SYSTEM CNV_LOOP_2_mess (* System Configuration *)
  (* Standard: 61499-1 *)
  (* Version 0.4, 2009-03-05, JHC, Holobloc Inc., Deleted Application. *)
  (* Version 0.3, 2003-12-05, JHC, Rockwell Automation, Renamed from NEWSYSTEM. *)
  (* Version 0.2, 2002-11-05, JHC, Rockwell Automation, Fixed missing (empty) FBD in Application. *)
  (* Version 0.1, 2002-01-17, JHC, Rockwell Automation, Minor cleanup *)
  (* Version 0.0, 2000-05-27, JHC, Rockwell Automation *)
  DEVICE HMI : FRAME_DEVICE(BOUNDS := [0,0,200,300], GRID := [10,10])
    RESOURCE CNV1_HMI : PANEL_RESOURCE
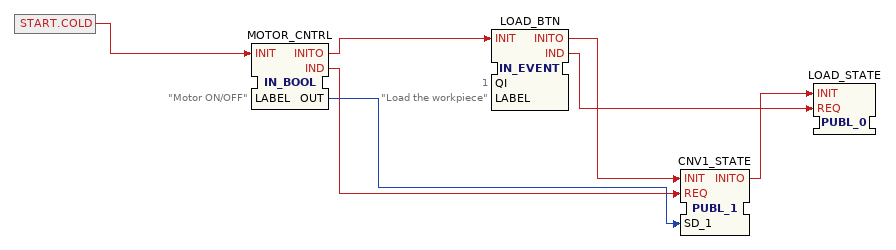
      FBS
        MOTOR_CNTRL : IN_BOOL(LABEL := "Motor ON/OFF");
        LOAD_BTN : IN_EVENT(QI := 1, LABEL := "Load the workpiece");
        LOAD_STATE : PUBL_0;
        CNV1_STATE : PUBL_1;
      END_FBS
      EVENT_CONNECTIONS
        START.COLD TO MOTOR_CNTRL.INIT;
        MOTOR_CNTRL.INITO TO LOAD_BTN.INIT;
        LOAD_BTN.INITO TO CNV1_STATE.INIT;
        CNV1_STATE.INITO TO LOAD_STATE.INIT;
        LOAD_BTN.IND TO LOAD_STATE.REQ;
        MOTOR_CNTRL.IND TO CNV1_STATE.REQ;
      END_CONNECTIONS
      DATA_CONNECTIONS
        MOTOR_CNTRL.OUT TO CNV1_STATE.SD_1;
      END_CONNECTIONS
    END_RESOURCE
  END_DEVICE
  DEVICE MODEL : FRAME_DEVICE(BOUNDS := [0,0,200,300])
    RESOURCE CNV1_MODEL : PANEL_RESOURCE
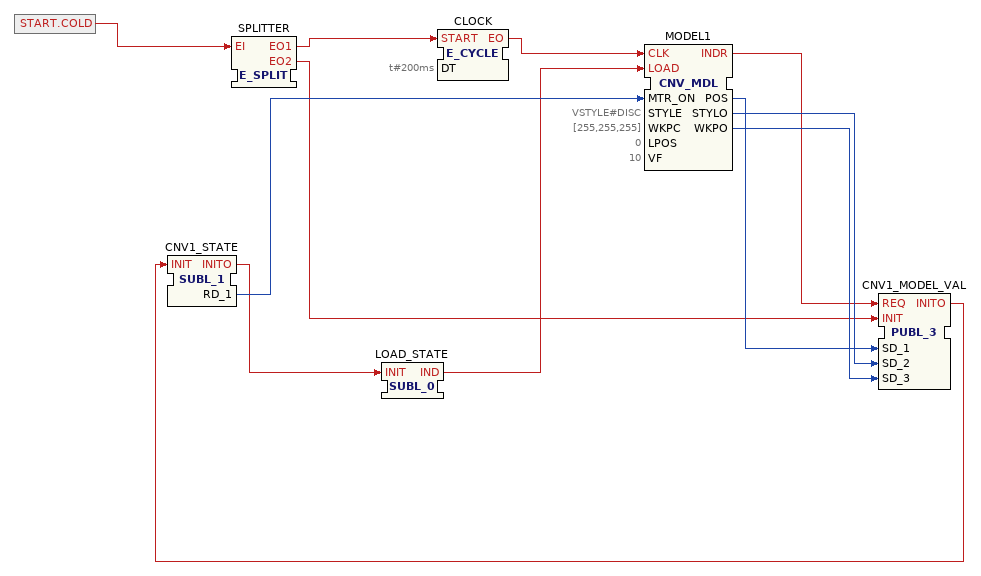
      FBS
        CLOCK : E_CYCLE(DT := t#200ms);
        MODEL1 : CNV_MDL(STYLE := VSTYLE#DISC, WKPC := [255,255,255], LPOS := 0, VF := 10);
        SPLITTER : E_SPLIT;
        CNV1_MODEL_VAL : PUBL_3;
        LOAD_STATE : SUBL_0;
        CNV1_STATE : SUBL_1;
      END_FBS
      EVENT_CONNECTIONS
        CLOCK.EO TO MODEL1.CLK;
        START.COLD TO SPLITTER.EI;
        SPLITTER.EO1 TO CLOCK.START;
        MODEL1.INDR TO CNV1_MODEL_VAL.REQ;
        SPLITTER.EO2 TO CNV1_MODEL_VAL.INIT;
        CNV1_MODEL_VAL.INITO TO CNV1_STATE.INIT;
        CNV1_STATE.INITO TO LOAD_STATE.INIT;
        LOAD_STATE.IND TO MODEL1.LOAD;
      END_CONNECTIONS
      DATA_CONNECTIONS
        MODEL1.POS TO CNV1_MODEL_VAL.SD_1;
        MODEL1.STYLO TO CNV1_MODEL_VAL.SD_2;
        MODEL1.WKPO TO CNV1_MODEL_VAL.SD_3;
        CNV1_STATE.RD_1 TO MODEL1.MTR_ON;
      END_CONNECTIONS
    END_RESOURCE
    RESOURCE CLK_MODEL : PANEL_RESOURCE
    END_RESOURCE
  END_DEVICE
  DEVICE VIEW : FRAME_DEVICE(BOUNDS := [200,0,300,300])
    RESOURCE VIEW_Resource : VIEW_PANEL(DIA := 20, SIZE := [15,15])
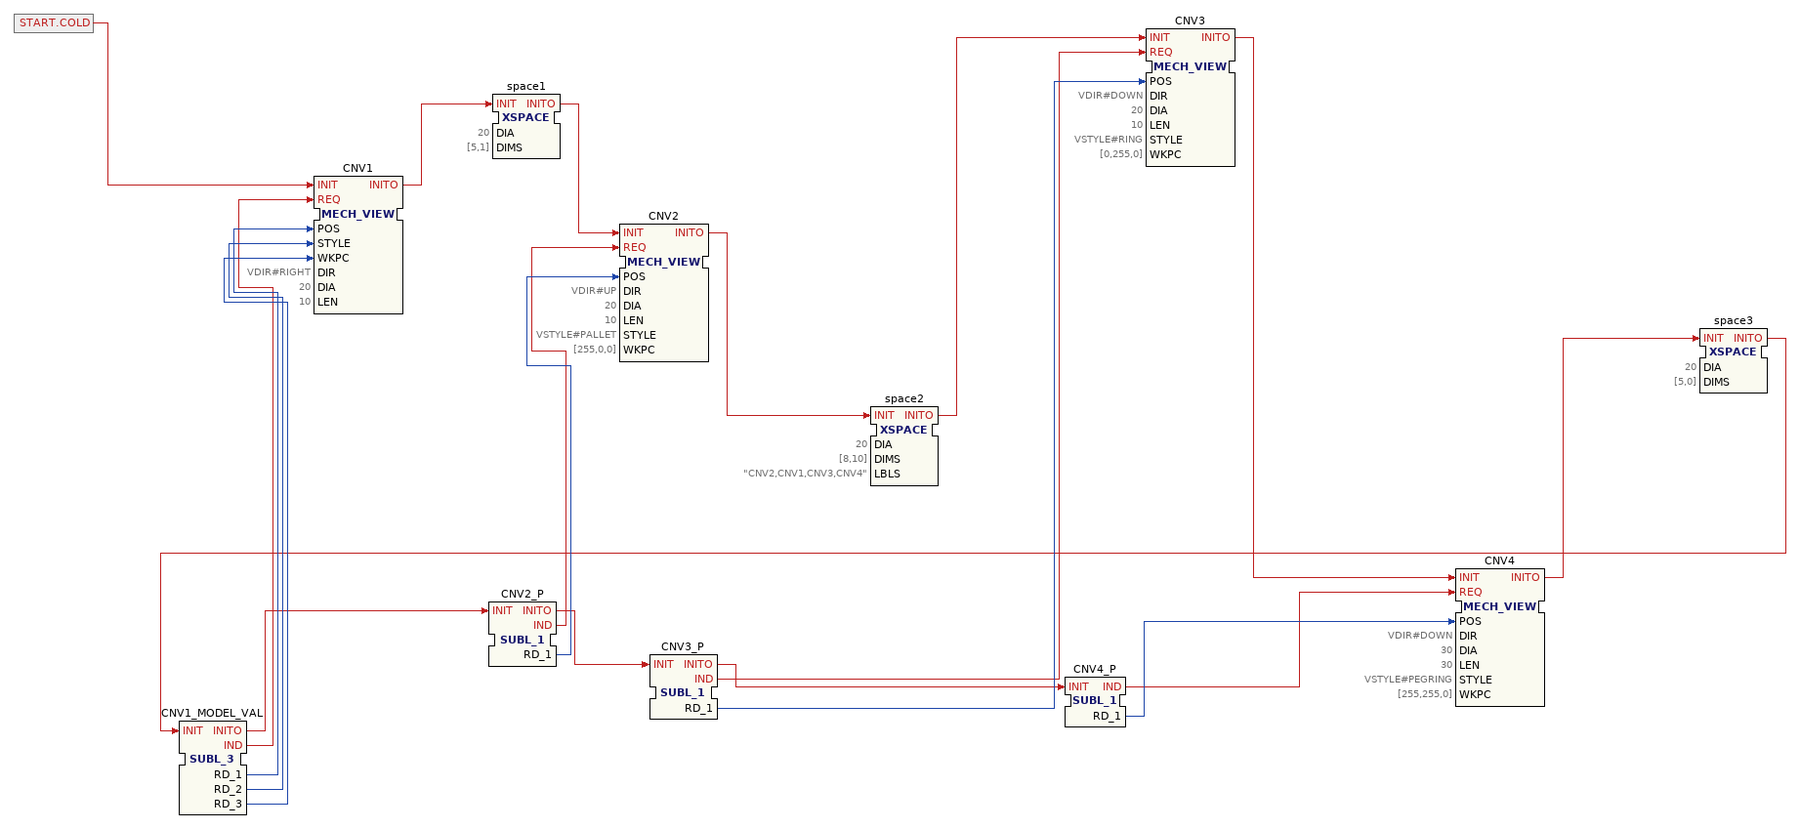
      FBS
        CNV1 : MECH_VIEW(DIR := VDIR#RIGHT, DIA := 20, LEN := 10);
        CNV2 : MECH_VIEW(DIR := VDIR#UP, DIA := 20, LEN := 10, STYLE := VSTYLE#PALLET, WKPC := [255,0,0]);
        CNV3 : MECH_VIEW(DIR := VDIR#DOWN, DIA := 20, LEN := 10, STYLE := VSTYLE#RING, WKPC := [0,255,0]);
        CNV4 : MECH_VIEW(DIR := VDIR#DOWN, DIA := 30, LEN := 30, STYLE := VSTYLE#PEGRING, WKPC := [255,255,0]);
        space1 : XSPACE(DIA := 20, DIMS := [5,1]);
        space2 : XSPACE(DIA := 20, DIMS := [8,10], LBLS := "CNV2,CNV1,CNV3,CNV4");
        space3 : XSPACE(DIA := 20, DIMS := [5,0]);
        CNV2_P : SUBL_1;
        CNV3_P : SUBL_1;
        CNV4_P : SUBL_1;
        CNV1_MODEL_VAL : SUBL_3;
      END_FBS
      EVENT_CONNECTIONS
        START.COLD TO CNV1.INIT;
        CNV3.INITO TO CNV4.INIT;
        CNV1.INITO TO space1.INIT;
        space1.INITO TO CNV2.INIT;
        CNV2.INITO TO space2.INIT;
        space2.INITO TO CNV3.INIT;
        CNV4.INITO TO space3.INIT;
        CNV2_P.INITO TO CNV3_P.INIT;
        CNV3_P.INITO TO CNV4_P.INIT;
        CNV2_P.IND TO CNV2.REQ;
        CNV3_P.IND TO CNV3.REQ;
        CNV4_P.IND TO CNV4.REQ;
        CNV1_MODEL_VAL.INITO TO CNV2_P.INIT;
        space3.INITO TO CNV1_MODEL_VAL.INIT;
        CNV1_MODEL_VAL.IND TO CNV1.REQ;
      END_CONNECTIONS
      DATA_CONNECTIONS
        CNV4_P.RD_1 TO CNV4.POS;
        CNV3_P.RD_1 TO CNV3.POS;
        CNV2_P.RD_1 TO CNV2.POS;
        CNV1_MODEL_VAL.RD_1 TO CNV1.POS;
        CNV1_MODEL_VAL.RD_2 TO CNV1.STYLE;
        CNV1_MODEL_VAL.RD_3 TO CNV1.WKPC;
      END_CONNECTIONS
    END_RESOURCE
  END_DEVICE
END_SYSTEM
